// TwinCAT 3 PLC project main
// ProgramVersion: 3.1.4024.0
// libraries:
//   Tc2_Standard, * (Beckhoff Automation GmbH)
//   Tc2_System, * (Beckhoff Automation GmbH)
//   Tc3_Module, * (Beckhoff Automation GmbH)
// project tree:
//   / GlobalTextList.TcGTLO, PlcTask.TcTTO, Visualization Manager.TcVMO (not stored)
//   POUs/ MAIN.TcPOU
//   VISUs/ Visu.TcVIS
// real-time tasks:
//   TASK PlcTask: cycle T#10ms, priority 20, ADS port 350

CONFIGURATION main
    RESOURCE PLC ON TwinCAT3
        TASK PlcTask(INTERVAL := T#10ms, PRIORITY := 20);
        PROGRAM MAIN WITH PlcTask : MAIN;
    END_RESOURCE
END_CONFIGURATION

// ---- POUs/MAIN.TcPOU
PROGRAM MAIN
VAR
	bS01 : BOOL;
	bS02 : BOOL;
	bQ01 : BOOL;
	bQ02 : BOOL;
END_VAR

bQ01 := (bS01 AND NOT bS02) OR (NOT bS01 AND NOT bS02);
bQ02 := (NOT bS01 AND bS02) OR (NOT bS01 AND NOT bS02);

END_PROGRAM

// ---- VISUs/Visu.TcVIS
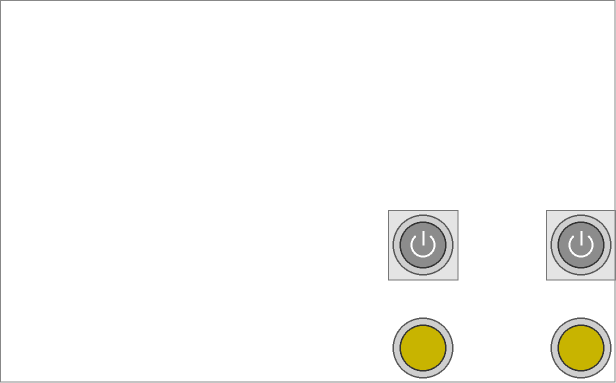
VISUALIZATION Visu  // 616x383
    PowerSwitch (388,210 70x70), variable: MAIN.bS01, behaviour: TOGGLE, style: Switch-PowerSwitch-Gray
    PowerSwitch (546,210 70x70), variable: MAIN.bS02, behaviour: TOGGLE, style: Switch-PowerSwitch-Gray
    Lamp1 (388,313 70x70), variable: MAIN.bQ01, style: Lamp-Lamp1-Yellow
    Lamp1 (546,313 70x70), variable: MAIN.bQ02, style: Lamp-Lamp1-Yellow
END_VISUALIZATION
